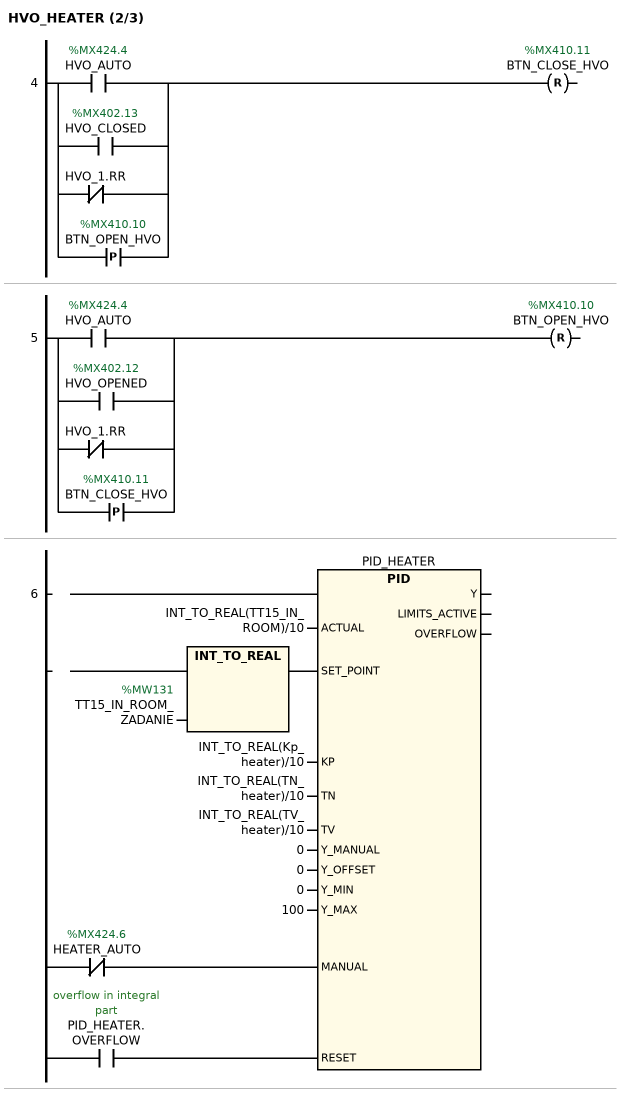
// NETWORK 4
//   HVO_AUTO: AT %MX424.4
//   HVO_CLOSED: AT %MX402.13
//   BTN_OPEN_HVO: AT %MX410.10
//   BTN_CLOSE_HVO: AT %MX410.11
_rt1(CLK := BTN_OPEN_HVO);
BTN_CLOSE_HVO R= HVO_AUTO OR HVO_CLOSED OR NOT HVO_1.RR OR _rt1.Q;

// NETWORK 5
//   HVO_AUTO: AT %MX424.4
//   HVO_OPENED: AT %MX402.12
//   BTN_CLOSE_HVO: AT %MX410.11
//   BTN_OPEN_HVO: AT %MX410.10
_rt2(CLK := BTN_CLOSE_HVO);
BTN_OPEN_HVO R= HVO_AUTO OR HVO_OPENED OR NOT HVO_1.RR OR _rt2.Q;

// NETWORK 6
//   TT15_IN_ROOM_ZADANIE: температура в комнате задание | AT %MW131
//   HEATER_AUTO: AT %MX424.6
//   PID_HEATER.OVERFLOW: overflow in integral part
PID_HEATER(
    ACTUAL := INT_TO_REAL(TT15_IN_ROOM)/10,
    SET_POINT := INT_TO_REAL(TT15_IN_ROOM_ZADANIE),
    KP := INT_TO_REAL(Kp_heater)/10,
    TN := INT_TO_REAL(TN_heater)/10,
    TV := INT_TO_REAL(TV_heater)/10,
    Y_MANUAL := 0,
    Y_OFFSET := 0,
    Y_MIN := 0,
    Y_MAX := 100,
    MANUAL := NOT HEATER_AUTO,
    RESET := PID_HEATER.OVERFLOW); // PID

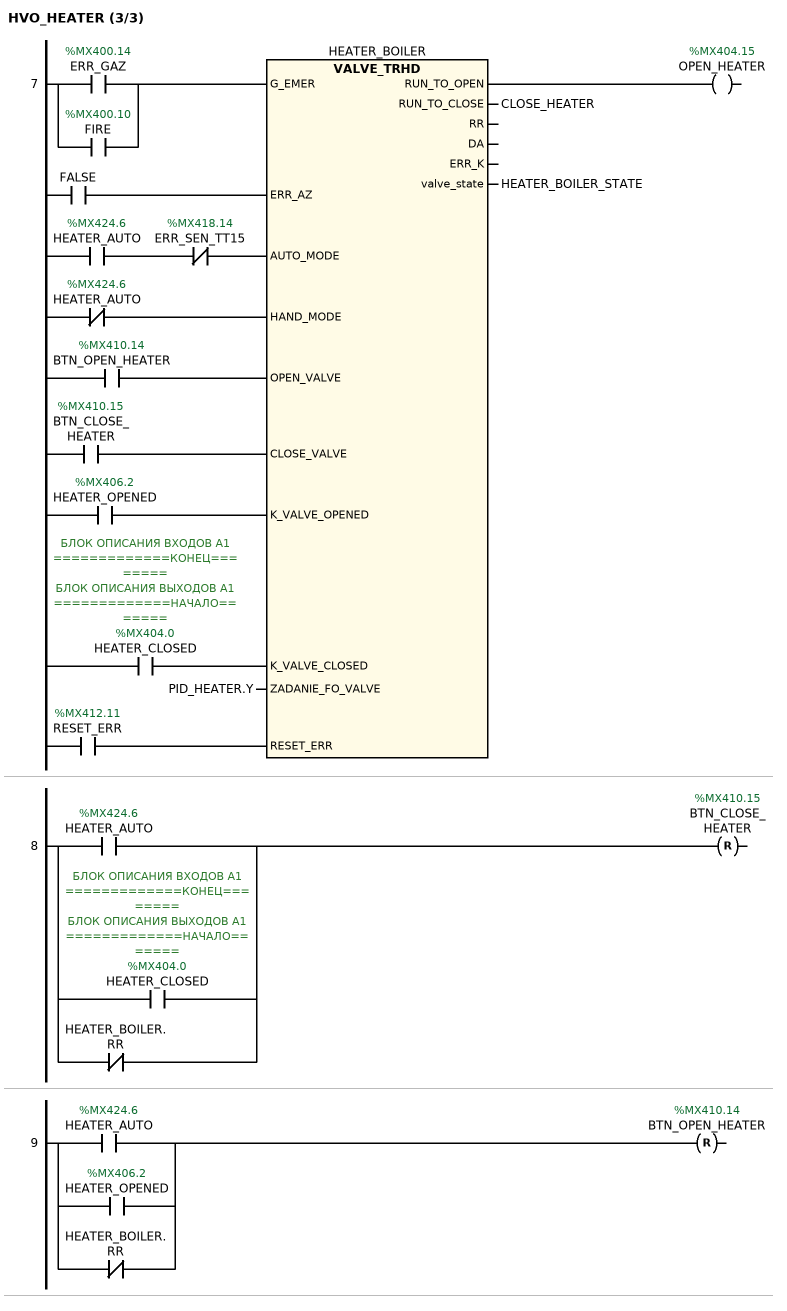
// NETWORK 7
//   ERR_GAZ: AT %MX400.14
//   FIRE: AT %MX400.10
//   HEATER_AUTO: AT %MX424.6
//   ERR_SEN_TT15: AT %MX418.14
//   BTN_OPEN_HEATER: AT %MX410.14
//   BTN_CLOSE_HEATER: AT %MX410.15
//   HEATER_OPENED: AT %MX406.2
//   HEATER_CLOSED: БЛОК ОПИСАНИЯ ВХОДОВ А1 =============КОНЕЦ======== БЛОК ОПИСАНИЯ ВЫХОДОВ А1 =============НАЧАЛО======= | AT %MX404.0
//   PID_HEATER.Y: manipulated variable, set value
//   RESET_ERR: AT %MX412.11
//   CLOSE_HEATER: AT %MX406.0
//   HEATER_BOILER_STATE: AT %MW404
//   OPEN_HEATER: AT %MX404.15
HEATER_BOILER(
    G_EMER := ERR_GAZ OR FIRE,
    ERR_AZ := FALSE,
    AUTO_MODE := HEATER_AUTO AND NOT ERR_SEN_TT15,
    HAND_MODE := NOT HEATER_AUTO,
    OPEN_VALVE := BTN_OPEN_HEATER,
    CLOSE_VALVE := BTN_CLOSE_HEATER,
    K_VALVE_OPENED := HEATER_OPENED,
    K_VALVE_CLOSED := HEATER_CLOSED,
    ZADANIE_FO_VALVE := PID_HEATER.Y,
    RESET_ERR := RESET_ERR,
    RUN_TO_CLOSE => CLOSE_HEATER,
    valve_state => HEATER_BOILER_STATE); // VALVE_TRHD
OPEN_HEATER := HEATER_BOILER.RUN_TO_OPEN;

// NETWORK 8
//   HEATER_AUTO: AT %MX424.6
//   HEATER_CLOSED: БЛОК ОПИСАНИЯ ВХОДОВ А1 =============КОНЕЦ======== БЛОК ОПИСАНИЯ ВЫХОДОВ А1 =============НАЧАЛО======= | AT %MX404.0
//   BTN_CLOSE_HEATER: AT %MX410.15
BTN_CLOSE_HEATER R= HEATER_AUTO OR HEATER_CLOSED OR NOT HEATER_BOILER.RR;

// NETWORK 9
//   HEATER_AUTO: AT %MX424.6
//   HEATER_OPENED: AT %MX406.2
//   BTN_OPEN_HEATER: AT %MX410.14
BTN_OPEN_HEATER R= HEATER_AUTO OR HEATER_OPENED OR NOT HEATER_BOILER.RR;

END_PROGRAM

// MyController/Application/FB/VALVE_TRHD
FUNCTION_BLOCK VALVE_TRHD
VAR_INPUT
	G_EMER: BOOL;
	ERR_AZ: BOOL;
	AUTO_MODE: BOOL;
	HAND_MODE: BOOL;
	OPEN_VALVE: BOOL;
	CLOSE_VALVE: BOOL;
	K_VALVE_OPENED: BOOL;
	K_VALVE_CLOSED: BOOL;
	ZADANIE_FO_VALVE: REAL;
	RESET_ERR: BOOL;	
END_VAR
VAR_OUTPUT
	RUN_TO_OPEN: BOOL;
	RUN_TO_CLOSE: BOOL;
	RR: BOOL;
	DA: BOOL;
	ERR_K: BOOL;
	valve_state: BYTE;
END_VAR
VAR
	TM_LT_VALVE: TON;
	RUN_VALVE_TO_OPEN: BOOL;
	CYCLE_OPEN: BOOL;
	CYCLE_CLOSE: BOOL;
END_VAR
VAR // added by the converter: edge detectors and wires of the graphical bodies
    _w1 : BOOL;
END_VAR

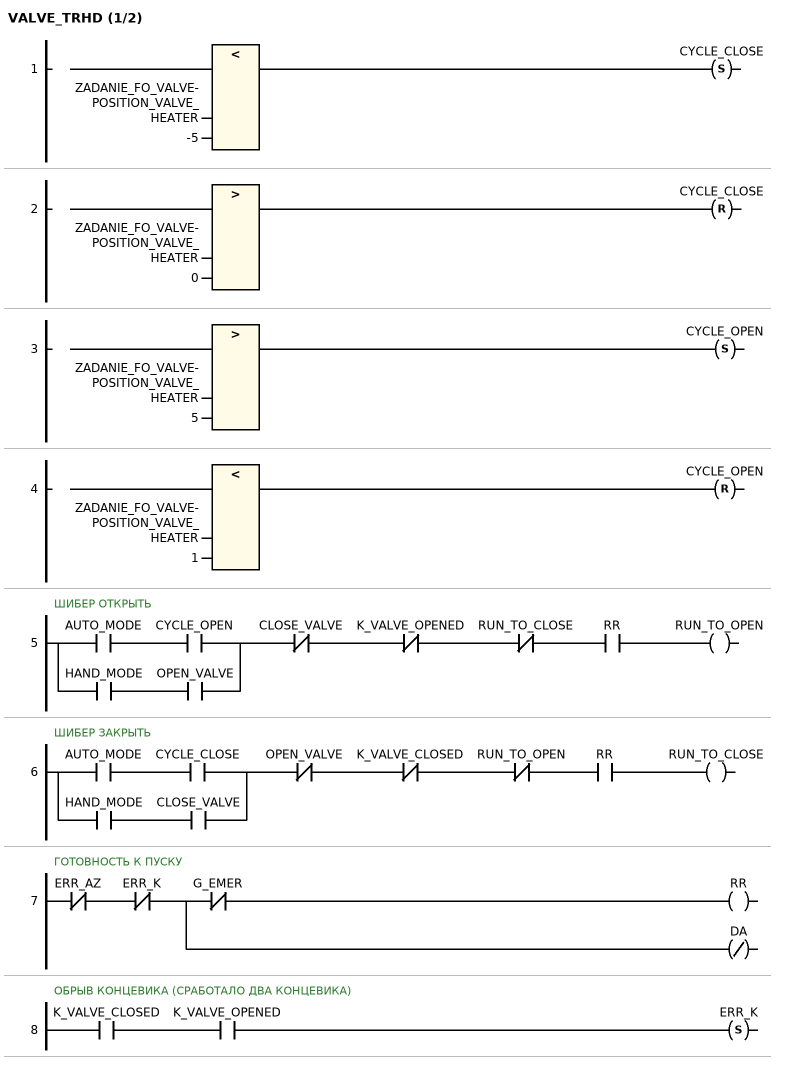
// NETWORK 1
CYCLE_CLOSE S= (ZADANIE_FO_VALVE-POSITION_VALVE_HEATER) < -5;

// NETWORK 2
CYCLE_CLOSE R= (ZADANIE_FO_VALVE-POSITION_VALVE_HEATER) > 0;

// NETWORK 3
CYCLE_OPEN S= (ZADANIE_FO_VALVE-POSITION_VALVE_HEATER) > 5;

// NETWORK 4
CYCLE_OPEN R= (ZADANIE_FO_VALVE-POSITION_VALVE_HEATER) < 1;

// NETWORK 5
// ШИБЕР ОТКРЫТЬ
RUN_TO_OPEN := (AUTO_MODE AND CYCLE_OPEN OR HAND_MODE AND OPEN_VALVE) AND NOT CLOSE_VALVE AND NOT K_VALVE_OPENED AND NOT RUN_TO_CLOSE AND RR;

// NETWORK 6
// ШИБЕР ЗАКРЫТЬ
RUN_TO_CLOSE := (AUTO_MODE AND CYCLE_CLOSE OR HAND_MODE AND CLOSE_VALVE) AND NOT OPEN_VALVE AND NOT K_VALVE_CLOSED AND NOT RUN_TO_OPEN AND RR;

// NETWORK 7
// ГОТОВНОСТЬ К ПУСКУ
_w1 := NOT ERR_AZ AND NOT ERR_K;
RR := _w1 AND NOT G_EMER;
DA := NOT _w1;

// NETWORK 8
// ОБРЫВ КОНЦЕВИКА (СРАБОТАЛО ДВА КОНЦЕВИКА)
ERR_K S= K_VALVE_CLOSED AND K_VALVE_OPENED;

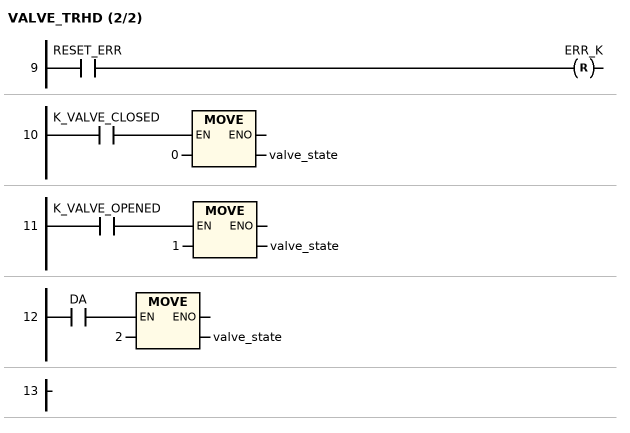
// NETWORK 9
ERR_K R= RESET_ERR;

// NETWORK 10
IF K_VALVE_CLOSED THEN valve_state := 0; END_IF

// NETWORK 11
IF K_VALVE_OPENED THEN valve_state := 1; END_IF

// NETWORK 12
IF DA THEN valve_state := 2; END_IF

// NETWORK 13

END_FUNCTION_BLOCK

// MyController/Application/connection
PROGRAM connection
VAR
	connection_off: TON;
	set_connection: BLINK;
	tm_connection: TON;
END_VAR
VAR // added by the converter: edge detectors and wires of the graphical bodies
    _rt1, _rt2 : R_TRIG;
END_VAR

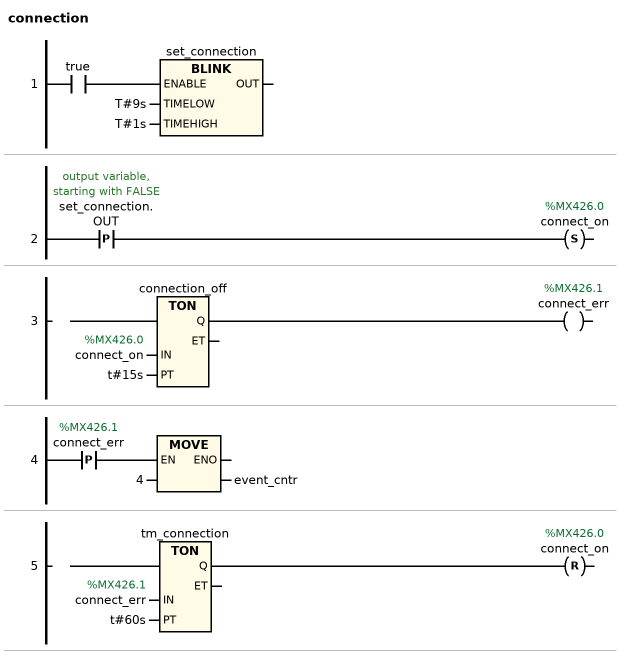
// NETWORK 1
set_connection(ENABLE := true, TIMELOW := T#9s, TIMEHIGH := T#1s); // BLINK

// NETWORK 2
//   set_connection.OUT: output variable, starting with FALSE
//   connect_on: AT %MX426.0
_rt1(CLK := set_connection.OUT);
connect_on S= _rt1.Q;

// NETWORK 3
//   connect_on: AT %MX426.0
//   connect_err: AT %MX426.1
connection_off(IN := connect_on, PT := t#15s); // TON
connect_err := connection_off.Q;

// NETWORK 4
//   connect_err: AT %MX426.1
//   event_cntr: AT %MW986
_rt2(CLK := connect_err);
IF _rt2.Q THEN event_cntr := 4; END_IF

// NETWORK 5
//   connect_err: AT %MX426.1
//   connect_on: AT %MX426.0
tm_connection(IN := connect_err, PT := t#60s); // TON
connect_on R= tm_connection.Q;

END_PROGRAM

// MyController/Application/DYMOHODS
PROGRAM DYMOHODS
VAR
	STOP_DYMOHOD_1: TON;
	STOP_DYMOHOD_2: TON;
END_VAR
VAR // added by the converter: edge detectors and wires of the graphical bodies
    _rt1, _rt2, _rt3, _rt4 : R_TRIG;
END_VAR

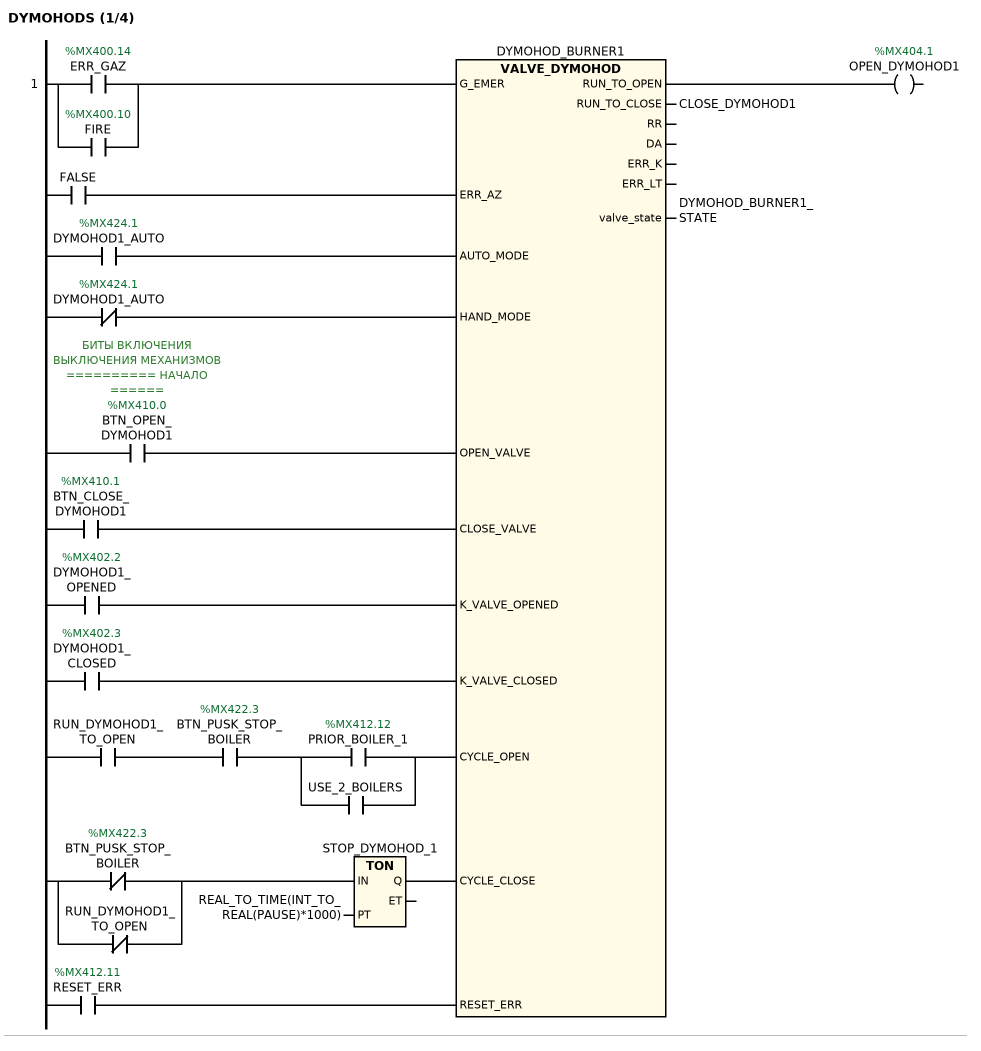
// NETWORK 1
//   ERR_GAZ: AT %MX400.14
//   FIRE: AT %MX400.10
//   DYMOHOD1_AUTO: AT %MX424.1
//   BTN_OPEN_DYMOHOD1: БИТЫ ВКЛЮЧЕНИЯ ВЫКЛЮЧЕНИЯ МЕХАНИЗМОВ ========== НАЧАЛО ====== | AT %MX410.0
//   BTN_CLOSE_DYMOHOD1: AT %MX410.1
//   DYMOHOD1_OPENED: AT %MX402.2
//   DYMOHOD1_CLOSED: AT %MX402.3
//   BTN_PUSK_STOP_BOILER: AT %MX422.3
//   PRIOR_BOILER_1: AT %MX412.12
//   RESET_ERR: AT %MX412.11
//   CLOSE_DYMOHOD1: AT %MX404.2
//   DYMOHOD_BURNER1_STATE: AT %MW401
//   OPEN_DYMOHOD1: AT %MX404.1
STOP_DYMOHOD_1(IN := NOT BTN_PUSK_STOP_BOILER OR NOT RUN_DYMOHOD1_TO_OPEN, PT := REAL_TO_TIME(INT_TO_REAL(PAUSE)*1000)); // TON
DYMOHOD_BURNER1(
    G_EMER := ERR_GAZ OR FIRE,
    ERR_AZ := FALSE,
    AUTO_MODE := DYMOHOD1_AUTO,
    HAND_MODE := NOT DYMOHOD1_AUTO,
    OPEN_VALVE := BTN_OPEN_DYMOHOD1,
    CLOSE_VALVE := BTN_CLOSE_DYMOHOD1,
    K_VALVE_OPENED := DYMOHOD1_OPENED,
    K_VALVE_CLOSED := DYMOHOD1_CLOSED,
    CYCLE_OPEN := RUN_DYMOHOD1_TO_OPEN AND BTN_PUSK_STOP_BOILER AND (PRIOR_BOILER_1 OR USE_2_BOILERS),
    CYCLE_CLOSE := STOP_DYMOHOD_1.Q,
    RESET_ERR := RESET_ERR,
    RUN_TO_CLOSE => CLOSE_DYMOHOD1,
    valve_state => DYMOHOD_BURNER1_STATE); // VALVE_DYMOHOD
OPEN_DYMOHOD1 := DYMOHOD_BURNER1.RUN_TO_OPEN;

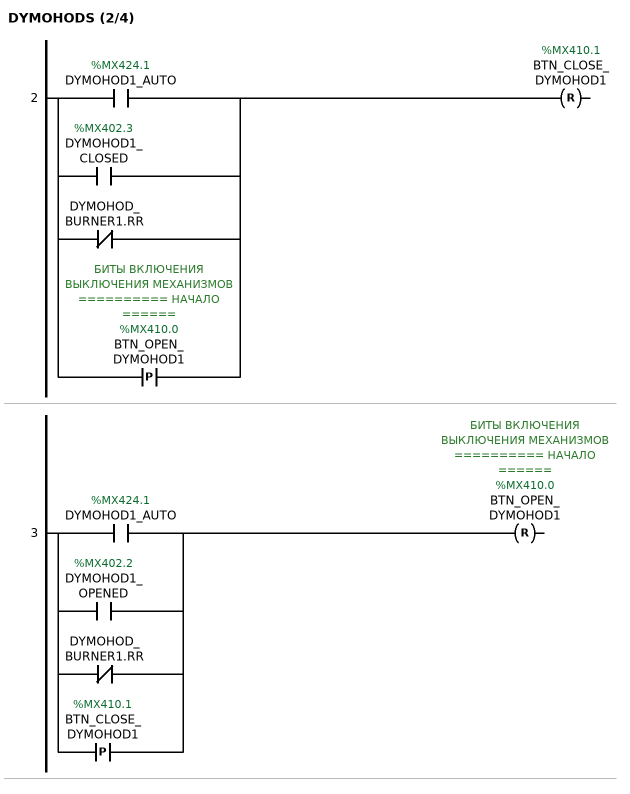
// NETWORK 2
//   DYMOHOD1_AUTO: AT %MX424.1
//   DYMOHOD1_CLOSED: AT %MX402.3
//   BTN_OPEN_DYMOHOD1: БИТЫ ВКЛЮЧЕНИЯ ВЫКЛЮЧЕНИЯ МЕХАНИЗМОВ ========== НАЧАЛО ====== | AT %MX410.0
//   BTN_CLOSE_DYMOHOD1: AT %MX410.1
_rt1(CLK := BTN_OPEN_DYMOHOD1);
BTN_CLOSE_DYMOHOD1 R= DYMOHOD1_AUTO OR DYMOHOD1_CLOSED OR NOT DYMOHOD_BURNER1.RR OR _rt1.Q;

// NETWORK 3
//   DYMOHOD1_AUTO: AT %MX424.1
//   DYMOHOD1_OPENED: AT %MX402.2
//   BTN_CLOSE_DYMOHOD1: AT %MX410.1
//   BTN_OPEN_DYMOHOD1: БИТЫ ВКЛЮЧЕНИЯ ВЫКЛЮЧЕНИЯ МЕХАНИЗМОВ ========== НАЧАЛО ====== | AT %MX410.0
_rt2(CLK := BTN_CLOSE_DYMOHOD1);
BTN_OPEN_DYMOHOD1 R= DYMOHOD1_AUTO OR DYMOHOD1_OPENED OR NOT DYMOHOD_BURNER1.RR OR _rt2.Q;

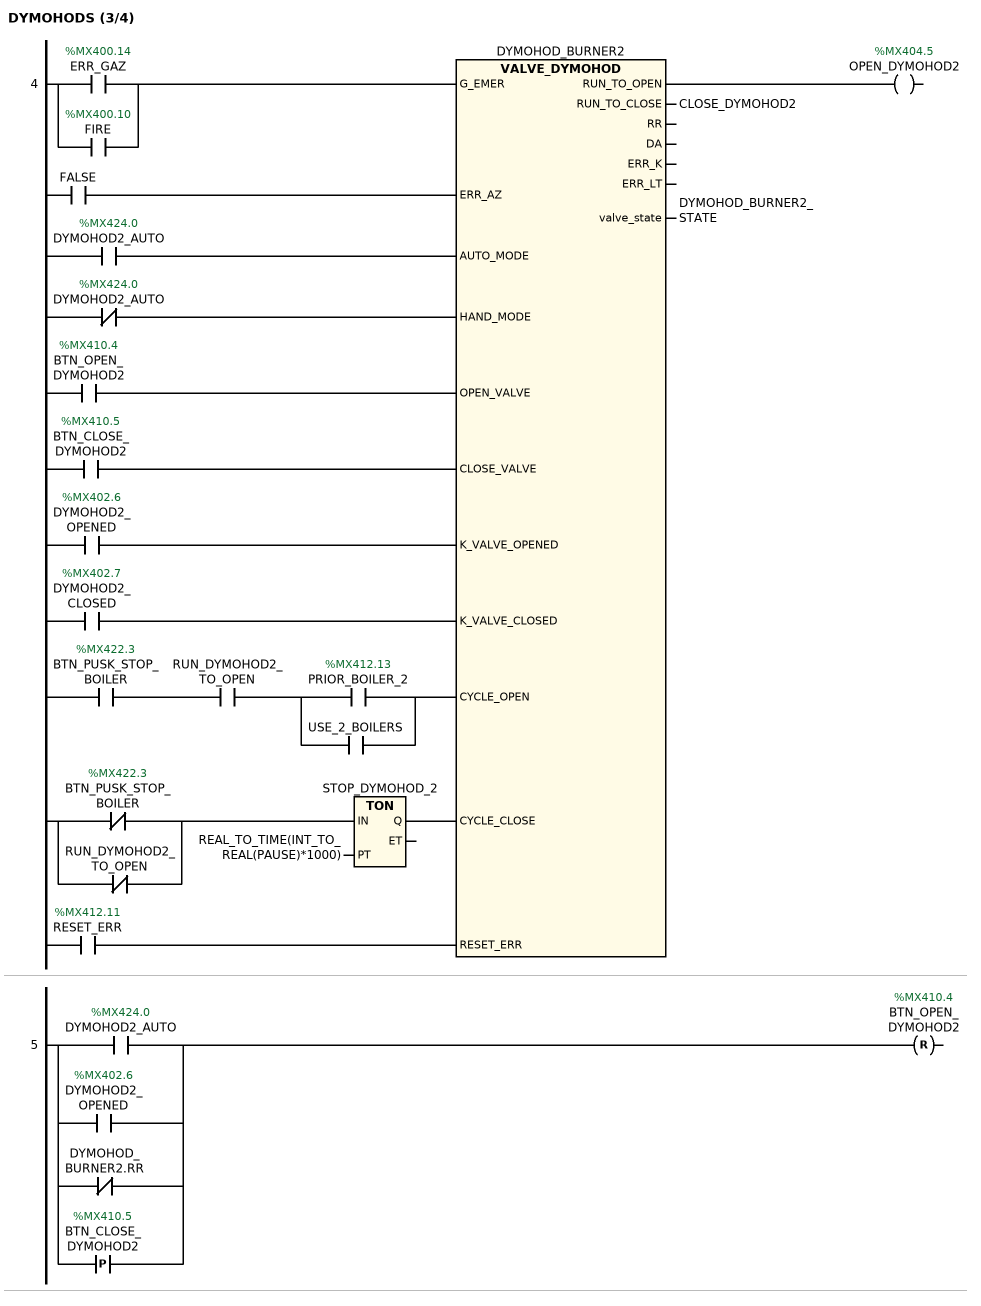
// NETWORK 4
//   ERR_GAZ: AT %MX400.14
//   FIRE: AT %MX400.10
//   DYMOHOD2_AUTO: AT %MX424.0
//   BTN_OPEN_DYMOHOD2: AT %MX410.4
//   BTN_CLOSE_DYMOHOD2: AT %MX410.5
//   DYMOHOD2_OPENED: AT %MX402.6
//   DYMOHOD2_CLOSED: AT %MX402.7
//   BTN_PUSK_STOP_BOILER: AT %MX422.3
//   PRIOR_BOILER_2: AT %MX412.13
//   RESET_ERR: AT %MX412.11
//   CLOSE_DYMOHOD2: AT %MX404.6
//   DYMOHOD_BURNER2_STATE: AT %MW402
//   OPEN_DYMOHOD2: AT %MX404.5
STOP_DYMOHOD_2(IN := NOT BTN_PUSK_STOP_BOILER OR NOT RUN_DYMOHOD2_TO_OPEN, PT := REAL_TO_TIME(INT_TO_REAL(PAUSE)*1000)); // TON
DYMOHOD_BURNER2(
    G_EMER := ERR_GAZ OR FIRE,
    ERR_AZ := FALSE,
    AUTO_MODE := DYMOHOD2_AUTO,
    HAND_MODE := NOT DYMOHOD2_AUTO,
    OPEN_VALVE := BTN_OPEN_DYMOHOD2,
    CLOSE_VALVE := BTN_CLOSE_DYMOHOD2,
    K_VALVE_OPENED := DYMOHOD2_OPENED,
    K_VALVE_CLOSED := DYMOHOD2_CLOSED,
    CYCLE_OPEN := BTN_PUSK_STOP_BOILER AND RUN_DYMOHOD2_TO_OPEN AND (PRIOR_BOILER_2 OR USE_2_BOILERS),
    CYCLE_CLOSE := STOP_DYMOHOD_2.Q,
    RESET_ERR := RESET_ERR,
    RUN_TO_CLOSE => CLOSE_DYMOHOD2,
    valve_state => DYMOHOD_BURNER2_STATE); // VALVE_DYMOHOD
OPEN_DYMOHOD2 := DYMOHOD_BURNER2.RUN_TO_OPEN;

// NETWORK 5
//   DYMOHOD2_AUTO: AT %MX424.0
//   DYMOHOD2_OPENED: AT %MX402.6
//   BTN_CLOSE_DYMOHOD2: AT %MX410.5
//   BTN_OPEN_DYMOHOD2: AT %MX410.4
_rt3(CLK := BTN_CLOSE_DYMOHOD2);
BTN_OPEN_DYMOHOD2 R= DYMOHOD2_AUTO OR DYMOHOD2_OPENED OR NOT DYMOHOD_BURNER2.RR OR _rt3.Q;

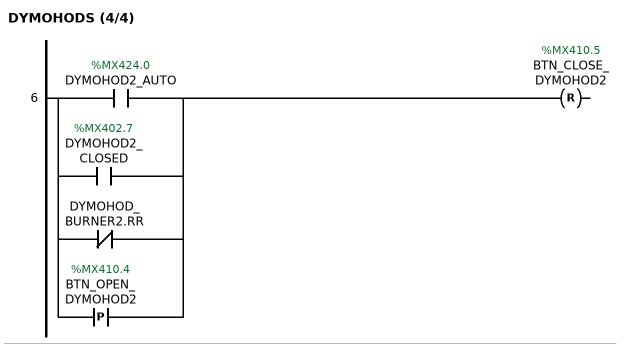
// NETWORK 6
//   DYMOHOD2_AUTO: AT %MX424.0
//   DYMOHOD2_CLOSED: AT %MX402.7
//   BTN_OPEN_DYMOHOD2: AT %MX410.4
//   BTN_CLOSE_DYMOHOD2: AT %MX410.5
_rt4(CLK := BTN_OPEN_DYMOHOD2);
BTN_CLOSE_DYMOHOD2 R= DYMOHOD2_AUTO OR DYMOHOD2_CLOSED OR NOT DYMOHOD_BURNER2.RR OR _rt4.Q;

END_PROGRAM

// MyController/Application/FB/VALVE_DYMOHOD
FUNCTION_BLOCK VALVE_DYMOHOD
VAR_INPUT
	G_EMER: BOOL;
	ERR_AZ: BOOL;
	AUTO_MODE: BOOL;
	HAND_MODE: BOOL;
	OPEN_VALVE: BOOL;
	CLOSE_VALVE: BOOL;
	K_VALVE_OPENED: BOOL;
	K_VALVE_CLOSED: BOOL;
	CYCLE_OPEN: BOOL;
	CYCLE_CLOSE: BOOL;
	RESET_ERR: BOOL;	
END_VAR
VAR_OUTPUT
	RUN_TO_OPEN: BOOL;
	RUN_TO_CLOSE: BOOL;
	RR: BOOL;
	DA: BOOL;
	ERR_K: BOOL;
	ERR_LT: BOOL;
	valve_state: BYTE;
END_VAR
VAR
	TM_LT_VALVE: TON;
END_VAR
VAR // added by the converter: edge detectors and wires of the graphical bodies
    _w1 : BOOL;
END_VAR

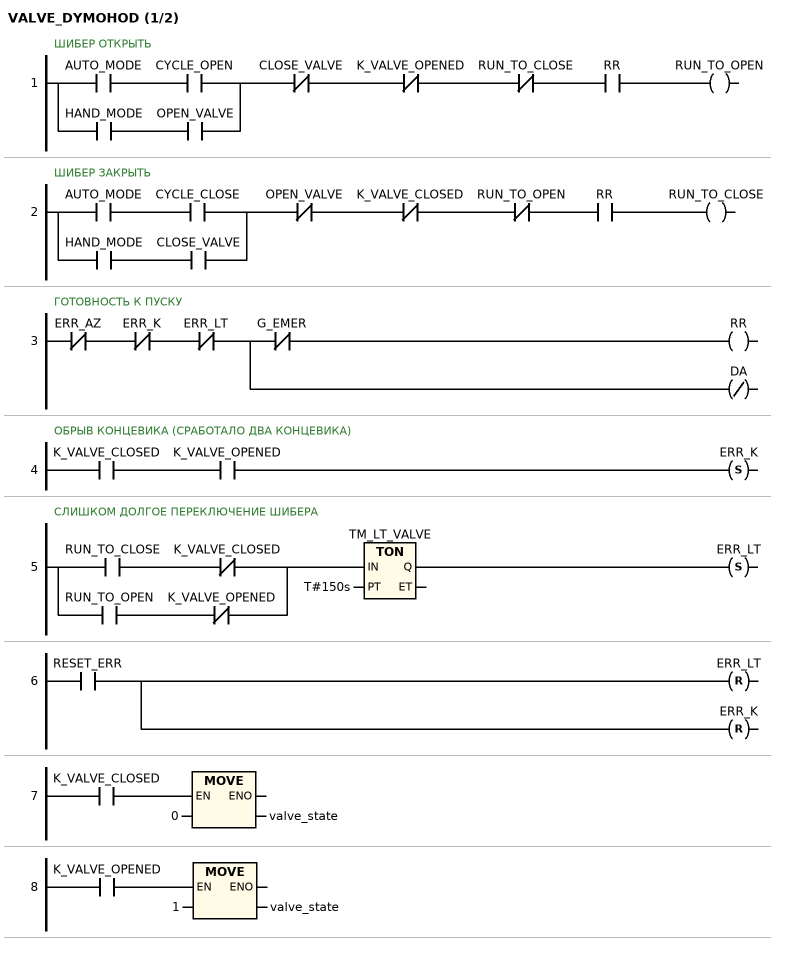
// NETWORK 1
// ШИБЕР ОТКРЫТЬ
RUN_TO_OPEN := (AUTO_MODE AND CYCLE_OPEN OR HAND_MODE AND OPEN_VALVE) AND NOT CLOSE_VALVE AND NOT K_VALVE_OPENED AND NOT RUN_TO_CLOSE AND RR;

// NETWORK 2
// ШИБЕР ЗАКРЫТЬ
RUN_TO_CLOSE := (AUTO_MODE AND CYCLE_CLOSE OR HAND_MODE AND CLOSE_VALVE) AND NOT OPEN_VALVE AND NOT K_VALVE_CLOSED AND NOT RUN_TO_OPEN AND RR;

// NETWORK 3
// ГОТОВНОСТЬ К ПУСКУ
_w1 := NOT ERR_AZ AND NOT ERR_K AND NOT ERR_LT;
RR := _w1 AND NOT G_EMER;
DA := NOT _w1;

// NETWORK 4
// ОБРЫВ КОНЦЕВИКА (СРАБОТАЛО ДВА КОНЦЕВИКА)
ERR_K S= K_VALVE_CLOSED AND K_VALVE_OPENED;

// NETWORK 5
// СЛИШКОМ ДОЛГОЕ ПЕРЕКЛЮЧЕНИЕ ШИБЕРА
TM_LT_VALVE(IN := RUN_TO_CLOSE AND NOT K_VALVE_CLOSED OR RUN_TO_OPEN AND NOT K_VALVE_OPENED, PT := T#150s); // TON
ERR_LT S= TM_LT_VALVE.Q;

// NETWORK 6
ERR_LT R= RESET_ERR;
ERR_K R= RESET_ERR;

// NETWORK 7
IF K_VALVE_CLOSED THEN valve_state := 0; END_IF

// NETWORK 8
IF K_VALVE_OPENED THEN valve_state := 1; END_IF

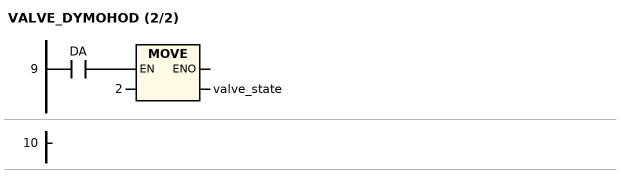
// NETWORK 9
IF DA THEN valve_state := 2; END_IF

// NETWORK 10

END_FUNCTION_BLOCK

// MyController/Application/RECIRCULATIONS_M5_M6_M7
PROGRAM RECIRCULATIONS_M5_M6_M7
VAR
	PUMP_M5_CYCLE: BOOL;
	PUMP_M6_CYCLE: BOOL;
	PUMP_M7_CYCLE: BOOL;
	PID_M7: PID;
END_VAR

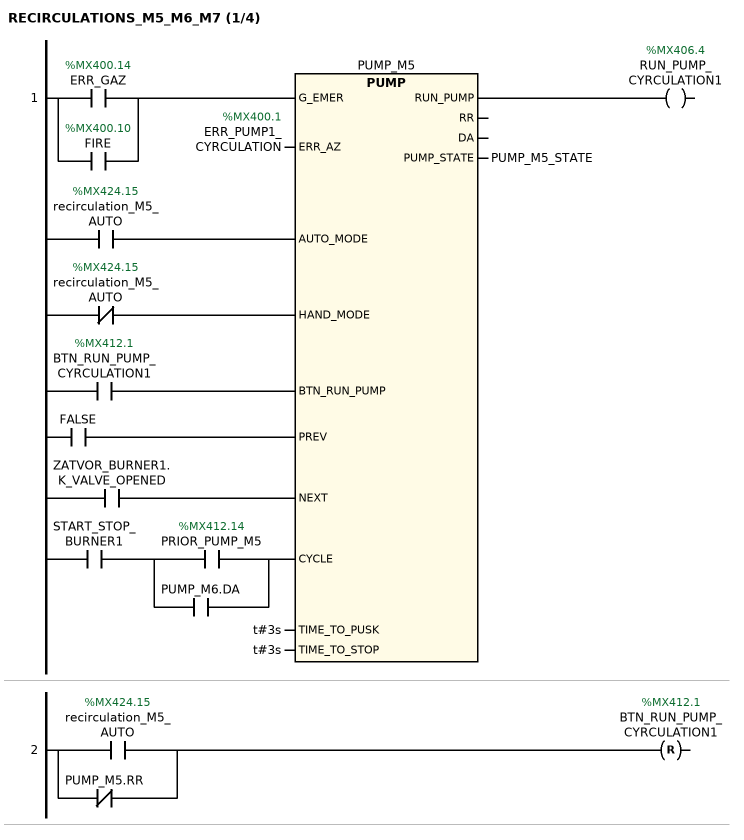
// NETWORK 1
//   ERR_GAZ: AT %MX400.14
//   FIRE: AT %MX400.10
//   ERR_PUMP1_CYRCULATION: AT %MX400.1
//   recirculation_M5_AUTO: AT %MX424.15
//   BTN_RUN_PUMP_CYRCULATION1: AT %MX412.1
//   PRIOR_PUMP_M5: AT %MX412.14
//   PUMP_M5_STATE: AT %MW413
//   RUN_PUMP_CYRCULATION1: AT %MX406.4
PUMP_M5(
    G_EMER := ERR_GAZ OR FIRE,
    ERR_AZ := ERR_PUMP1_CYRCULATION,
    AUTO_MODE := recirculation_M5_AUTO,
    HAND_MODE := NOT recirculation_M5_AUTO,
    BTN_RUN_PUMP := BTN_RUN_PUMP_CYRCULATION1,
    PREV := FALSE,
    NEXT := ZATVOR_BURNER1.K_VALVE_OPENED,
    CYCLE := START_STOP_BURNER1 AND (PRIOR_PUMP_M5 OR PUMP_M6.DA),
    TIME_TO_PUSK := t#3s,
    TIME_TO_STOP := t#3s,
    PUMP_STATE => PUMP_M5_STATE); // PUMP
RUN_PUMP_CYRCULATION1 := PUMP_M5.RUN_PUMP;

// NETWORK 2
//   recirculation_M5_AUTO: AT %MX424.15
//   BTN_RUN_PUMP_CYRCULATION1: AT %MX412.1
BTN_RUN_PUMP_CYRCULATION1 R= recirculation_M5_AUTO OR NOT PUMP_M5.RR;

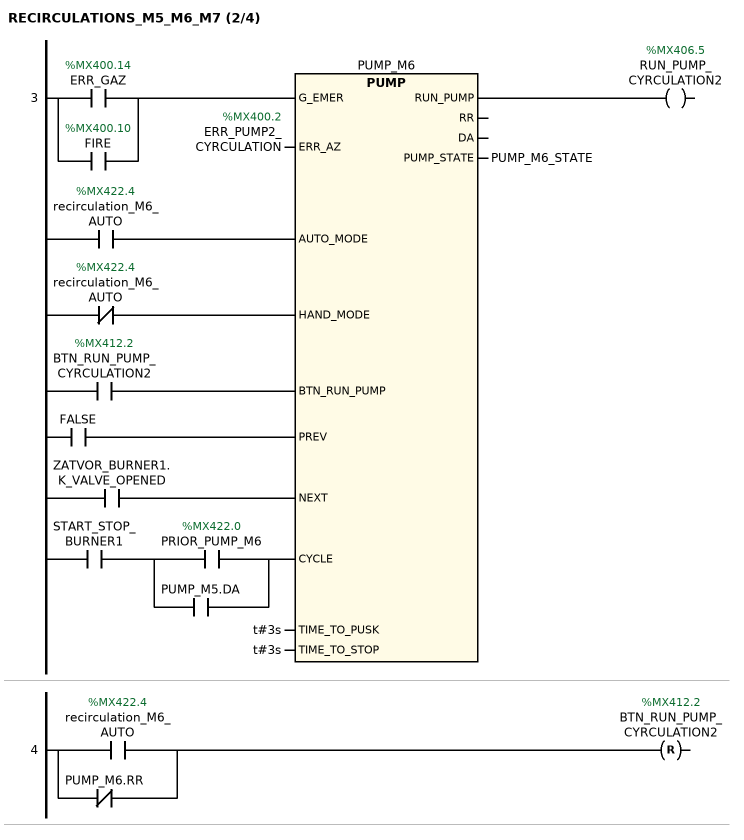
// NETWORK 3
//   ERR_GAZ: AT %MX400.14
//   FIRE: AT %MX400.10
//   ERR_PUMP2_CYRCULATION: AT %MX400.2
//   recirculation_M6_AUTO: AT %MX422.4
//   BTN_RUN_PUMP_CYRCULATION2: AT %MX412.2
//   PRIOR_PUMP_M6: AT %MX422.0
//   PUMP_M6_STATE: AT %MW414
//   RUN_PUMP_CYRCULATION2: AT %MX406.5
PUMP_M6(
    G_EMER := ERR_GAZ OR FIRE,
    ERR_AZ := ERR_PUMP2_CYRCULATION,
    AUTO_MODE := recirculation_M6_AUTO,
    HAND_MODE := NOT recirculation_M6_AUTO,
    BTN_RUN_PUMP := BTN_RUN_PUMP_CYRCULATION2,
    PREV := FALSE,
    NEXT := ZATVOR_BURNER1.K_VALVE_OPENED,
    CYCLE := START_STOP_BURNER1 AND (PRIOR_PUMP_M6 OR PUMP_M5.DA),
    TIME_TO_PUSK := t#3s,
    TIME_TO_STOP := t#3s,
    PUMP_STATE => PUMP_M6_STATE); // PUMP
RUN_PUMP_CYRCULATION2 := PUMP_M6.RUN_PUMP;

// NETWORK 4
//   recirculation_M6_AUTO: AT %MX422.4
//   BTN_RUN_PUMP_CYRCULATION2: AT %MX412.2
BTN_RUN_PUMP_CYRCULATION2 R= recirculation_M6_AUTO OR NOT PUMP_M6.RR;

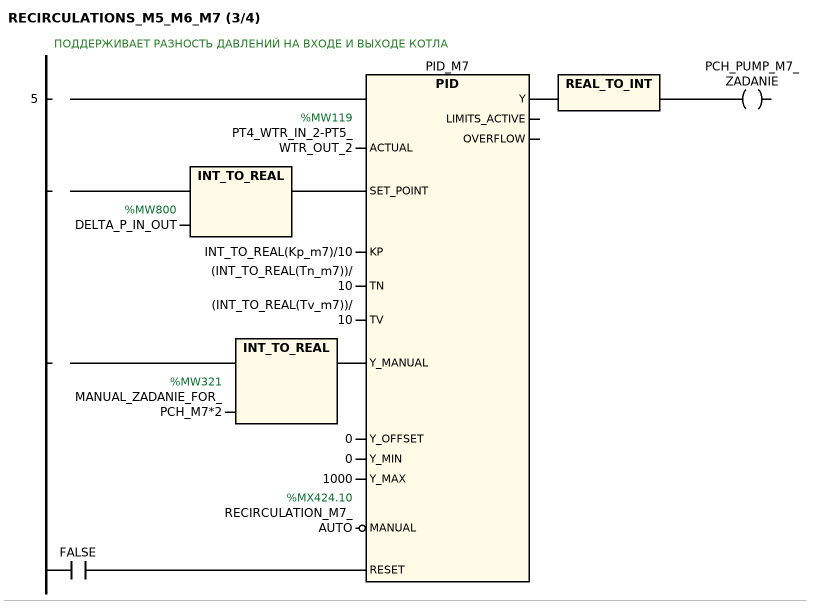
// NETWORK 5
// ПОДДЕРЖИВАЕТ РАЗНОСТЬ ДАВЛЕНИЙ НА ВХОДЕ И ВЫХОДЕ КОТЛА
//   PT4_WTR_IN_2-PT5_WTR_OUT_2: AT %MW119
//   DELTA_P_IN_OUT: AT %MW800
//   MANUAL_ZADANIE_FOR_PCH_M7*2: AT %MW321
//   RECIRCULATION_M7_AUTO: AT %MX424.10
PID_M7(
    ACTUAL := PT4_WTR_IN_2-PT5_WTR_OUT_2,
    SET_POINT := INT_TO_REAL(DELTA_P_IN_OUT),
    KP := INT_TO_REAL(Kp_m7)/10,
    TN := (INT_TO_REAL(Tn_m7))/10,
    TV := (INT_TO_REAL(Tv_m7))/10,
    Y_MANUAL := INT_TO_REAL(MANUAL_ZADANIE_FOR_PCH_M7*2),
    Y_OFFSET := 0,
    Y_MIN := 0,
    Y_MAX := 1000,
    MANUAL := NOT RECIRCULATION_M7_AUTO,
    RESET := FALSE); // PID
PCH_PUMP_M7_ZADANIE := REAL_TO_INT(PID_M7.Y);

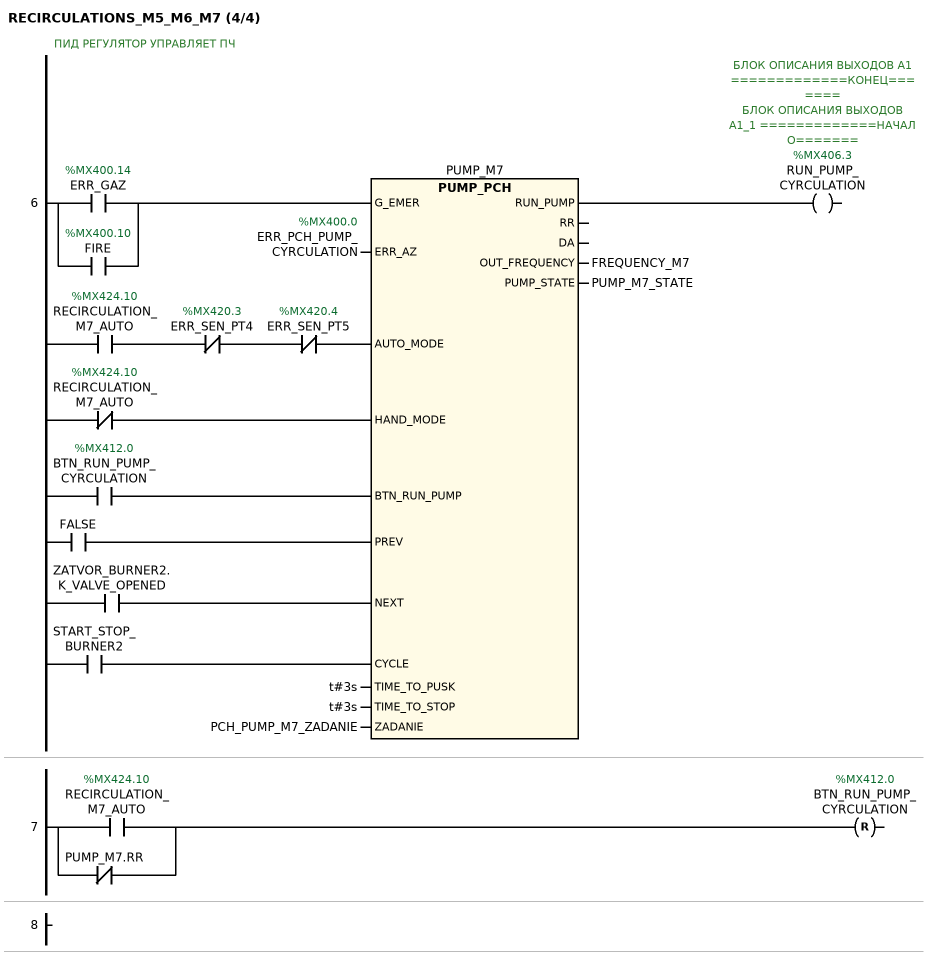
// NETWORK 6
// ПИД РЕГУЛЯТОР УПРАВЛЯЕТ ПЧ
//   ERR_GAZ: AT %MX400.14
//   FIRE: AT %MX400.10
//   ERR_PCH_PUMP_CYRCULATION: БЛОК ДЛЯ ОБМЕНА С ОВЕНОМ ======КОЕЦ====== БЛОК ОПИСАНИЯ ВХОДОВ А1_1 A1_2 =============НАЧАЛО======= | AT %MX400.0
//   RECIRCULATION_M7_AUTO: AT %MX424.10
//   ERR_SEN_PT4: AT %MX420.3
//   ERR_SEN_PT5: AT %MX420.4
//   BTN_RUN_PUMP_CYRCULATION: AT %MX412.0
//   FREQUENCY_M7: AT %MW136
//   PUMP_M7_STATE: AT %MW415
//   RUN_PUMP_CYRCULATION: БЛОК ОПИСАНИЯ ВЫХОДОВ А1 =============КОНЕЦ======= БЛОК ОПИСАНИЯ ВЫХОДОВ А1_1 =============НАЧАЛО======= | AT %MX406.3
PUMP_M7(
    G_EMER := ERR_GAZ OR FIRE,
    ERR_AZ := ERR_PCH_PUMP_CYRCULATION,
    AUTO_MODE := RECIRCULATION_M7_AUTO AND NOT ERR_SEN_PT4 AND NOT ERR_SEN_PT5,
    HAND_MODE := NOT RECIRCULATION_M7_AUTO,
    BTN_RUN_PUMP := BTN_RUN_PUMP_CYRCULATION,
    PREV := FALSE,
    NEXT := ZATVOR_BURNER2.K_VALVE_OPENED,
    CYCLE := START_STOP_BURNER2,
    TIME_TO_PUSK := t#3s,
    TIME_TO_STOP := t#3s,
    ZADANIE := PCH_PUMP_M7_ZADANIE,
    OUT_FREQUENCY => FREQUENCY_M7,
    PUMP_STATE => PUMP_M7_STATE); // PUMP_PCH
RUN_PUMP_CYRCULATION := PUMP_M7.RUN_PUMP;

// NETWORK 7
//   RECIRCULATION_M7_AUTO: AT %MX424.10
//   BTN_RUN_PUMP_CYRCULATION: AT %MX412.0
BTN_RUN_PUMP_CYRCULATION R= RECIRCULATION_M7_AUTO OR NOT PUMP_M7.RR;

// NETWORK 8

END_PROGRAM

// MyController/Application/FB/PUMP
FUNCTION_BLOCK PUMP
VAR_INPUT
	G_EMER: BOOL;
	ERR_AZ: BOOL;		
	AUTO_MODE: BOOL;
	HAND_MODE: BOOL;
	BTN_RUN_PUMP: BOOL;
	PREV: BOOL;
	NEXT: BOOL;	
	CYCLE: BOOL;	
	TIME_TO_PUSK: TIME;
	TIME_TO_STOP: TIME;		
END_VAR
VAR_OUTPUT
	RUN_PUMP: BOOL;
	RR: BOOL;
	DA: BOOL;	
	PUMP_STATE: BYTE;
END_VAR
VAR
	AUTO: BOOL;
	TM_PUSK_PUMP: TON;
	TM_STOP_PUMP: TON;
END_VAR
VAR // added by the converter: edge detectors and wires of the graphical bodies
    _w1 : BOOL;
END_VAR

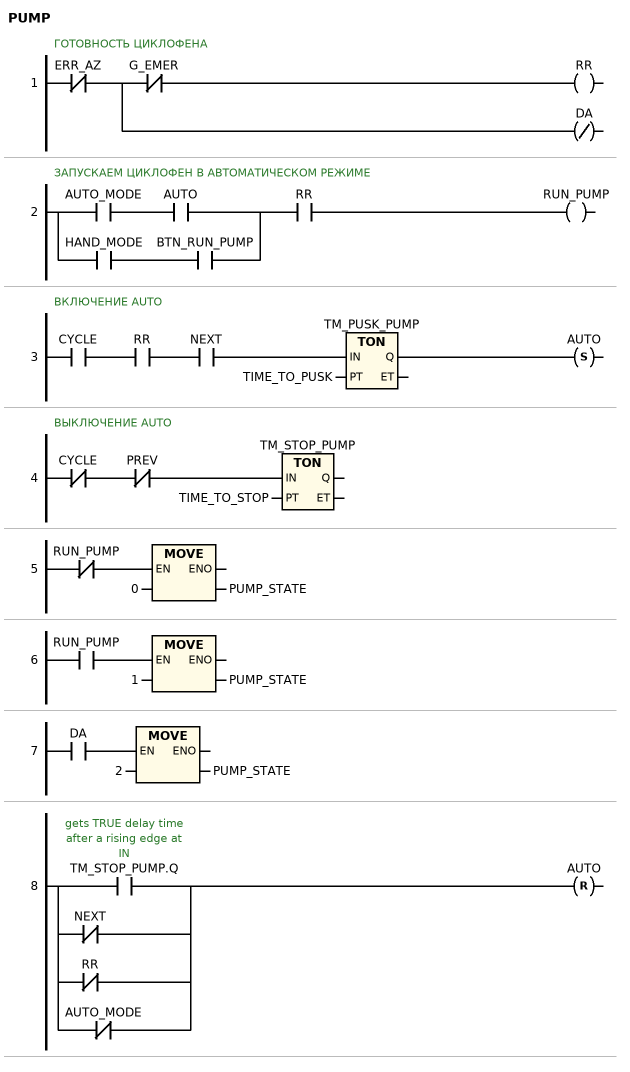
// NETWORK 1
// ГОТОВНОСТЬ ЦИКЛОФЕНА
_w1 := NOT ERR_AZ;
RR := _w1 AND NOT G_EMER;
DA := NOT _w1;

// NETWORK 2
// ЗАПУСКАЕМ ЦИКЛОФЕН В АВТОМАТИЧЕСКОМ РЕЖИМЕ
RUN_PUMP := (AUTO_MODE AND AUTO OR HAND_MODE AND BTN_RUN_PUMP) AND RR;

// NETWORK 3
// ВКЛЮЧЕНИЕ AUTO
TM_PUSK_PUMP(IN := CYCLE AND RR AND NEXT, PT := TIME_TO_PUSK); // TON
AUTO S= TM_PUSK_PUMP.Q;

// NETWORK 4
// ВЫКЛЮЧЕНИЕ AUTO
TM_STOP_PUMP(IN := NOT CYCLE AND NOT PREV, PT := TIME_TO_STOP); // TON

// NETWORK 5
IF NOT RUN_PUMP THEN PUMP_STATE := 0; END_IF

// NETWORK 6
IF RUN_PUMP THEN PUMP_STATE := 1; END_IF

// NETWORK 7
IF DA THEN PUMP_STATE := 2; END_IF

// NETWORK 8
//   TM_STOP_PUMP.Q: gets TRUE delay time after a rising edge at IN
AUTO R= TM_STOP_PUMP.Q OR NOT NEXT OR NOT RR OR NOT AUTO_MODE;

END_FUNCTION_BLOCK

// MyController/Application/FB/PUMP_PCH
FUNCTION_BLOCK PUMP_PCH
VAR_INPUT
	G_EMER: BOOL;
	ERR_AZ: BOOL;		
	AUTO_MODE: BOOL;
	HAND_MODE: BOOL;
	BTN_RUN_PUMP: BOOL;
	PREV: BOOL;
	NEXT: BOOL;	
	CYCLE: BOOL;	
	TIME_TO_PUSK: TIME;
	TIME_TO_STOP: TIME;		
	ZADANIE: INT;
END_VAR
VAR_OUTPUT
	RUN_PUMP: BOOL;
	RR: BOOL;
	DA: BOOL;	
	OUT_FREQUENCY: INT;
	PUMP_STATE: BYTE;
END_VAR
VAR
	AUTO: BOOL;
	TM_PUSK_PUMP: TON;
	TM_STOP_PUMP: TON;
END_VAR
VAR // added by the converter: edge detectors and wires of the graphical bodies
    _w1 : BOOL;
END_VAR

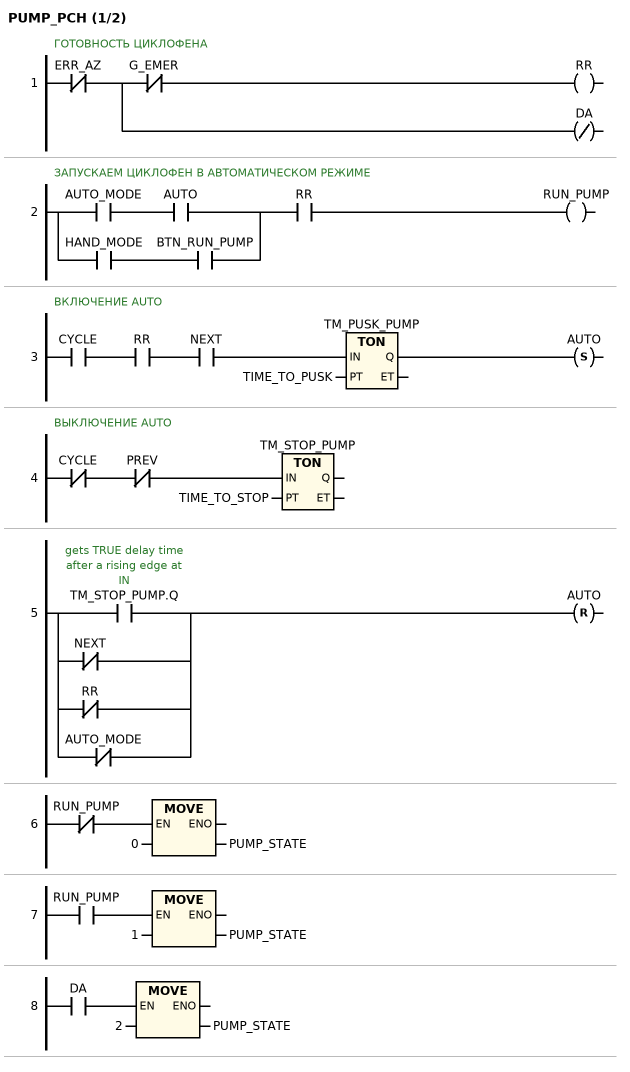
// NETWORK 1
// ГОТОВНОСТЬ ЦИКЛОФЕНА
_w1 := NOT ERR_AZ;
RR := _w1 AND NOT G_EMER;
DA := NOT _w1;

// NETWORK 2
// ЗАПУСКАЕМ ЦИКЛОФЕН В АВТОМАТИЧЕСКОМ РЕЖИМЕ
RUN_PUMP := (AUTO_MODE AND AUTO OR HAND_MODE AND BTN_RUN_PUMP) AND RR;

// NETWORK 3
// ВКЛЮЧЕНИЕ AUTO
TM_PUSK_PUMP(IN := CYCLE AND RR AND NEXT, PT := TIME_TO_PUSK); // TON
AUTO S= TM_PUSK_PUMP.Q;

// NETWORK 4
// ВЫКЛЮЧЕНИЕ AUTO
TM_STOP_PUMP(IN := NOT CYCLE AND NOT PREV, PT := TIME_TO_STOP); // TON

// NETWORK 5
//   TM_STOP_PUMP.Q: gets TRUE delay time after a rising edge at IN
AUTO R= TM_STOP_PUMP.Q OR NOT NEXT OR NOT RR OR NOT AUTO_MODE;

// NETWORK 6
IF NOT RUN_PUMP THEN PUMP_STATE := 0; END_IF

// NETWORK 7
IF RUN_PUMP THEN PUMP_STATE := 1; END_IF

// NETWORK 8
IF DA THEN PUMP_STATE := 2; END_IF

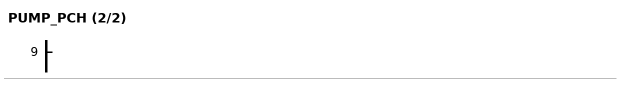
// NETWORK 9

END_FUNCTION_BLOCK

// MyController/Application/POUWER_BOILER
PROGRAM POUWER_BOILER
VAR
	BLINK_RESET_FLOW : BLINK;
	RISE_IMPUT_FLOW : R_TRIG;
	good: BOOL;
	K: REAL;
	TF: REAL;
	POWER_BURNER: REAL;
	//power_utilizator: REAL;
END_VAR

POWER_GRAFIC:=FLOW_GRAFIC*(TMP_PODACHA-TMP_OBRATKA)*99.82/1000000;//Определяем мощность расчетную для котлов

BLINK_RESET_FLOW(ENABLE:=1,TIMELOW:=T#9S,TIMEHIGH:=T#1S);
RISE_IMPUT_FLOW(CLK:=BLINK_RESET_FLOW.OUT);
IF reset_flowmetr.zero_flow=0 AND RISE_IMPUT_FLOW.Q=1 THEN
	power_utilizator:=power_utilizator+FLOW_BOILER_2*(TT7_WTR_IN_2-TT6_WTR_UTIL_IN)*99.82/1000000/360;
END_IF

//fl_g_s:=Qb_s;
//fl_g_l:=Qb_l;
flow_gaz:=Qb_l;
flow_gaz:=SHL(flow_gaz,16);
flow_gaz:=flow_gaz+Qb_s;
V_gaz:=Vb_l;
V_gaz:=SHL(V_gaz,16);
V_gaz:=V_gaz+Vb_s;
//flow_gaz:=flow_gaz*65636;


//	POWER_BOILER_1:=FLOW_BOILER_1*(TT3_WTR_OUT_1-TT2_WTR_IN_1)*99.82/1000000;
//	POWER_BOILER_2:=FLOW_BOILER_2*(TT8_WTR_OUT_2-TT7_WTR_IN_2)*99.82/1000000;

//T_ZADANNOE:= ((POWER_GRAFIC + TT2_WTR_IN_1*(FLOW_BOILER_1+FLOW_BOILER_2))/FLOW_BOILER_1+FLOW_BOILER_2)*(K+(T1_GRAFIC-TF));

//TEMP_POROG_2:= REAL_TO_INT(T_ZADANNOE);

//IF PRIOR_BOILER_1 
//	THEN POWER_BURNER:=1000;
//	ELSE POWER_BURNER:=800;
//END_IF

//POWER_GRAFIC:=FLOW_GRAFIC*(TMP_PODACHA-TMP_OBRATKA);//Определяем мощность расчетную для котлов

//IF POWER_GRAFIC > POWER_BURNER

IF MEDIUM_TEMP_AIR<tmp_use_1_and_2_boiler/10 OR POWER_GRAFIC>=0.95*POWER_BOILER2/1000
	THEN USE_2_BOILERS:=1;
	ELSE USE_2_BOILERS:=0;
END_IF

END_PROGRAM

// MyController/Application/ALL_ERR
PROGRAM ALL_ERR
VAR
	DA_ALL_1: BOOL;
	DA_ALL_2: BOOL;
	DA_ALL_3: BOOL;
	DA_ALL_4: BOOL;
	DA_ALL_5: BOOL;
	DA_ALL_6: BOOL;
	DA_ALL_7: BOOL;
	DA_ALL_8: BOOL;
	DA_ALL_9: BOOL;
	DA_ALL_10: BOOL;
END_VAR

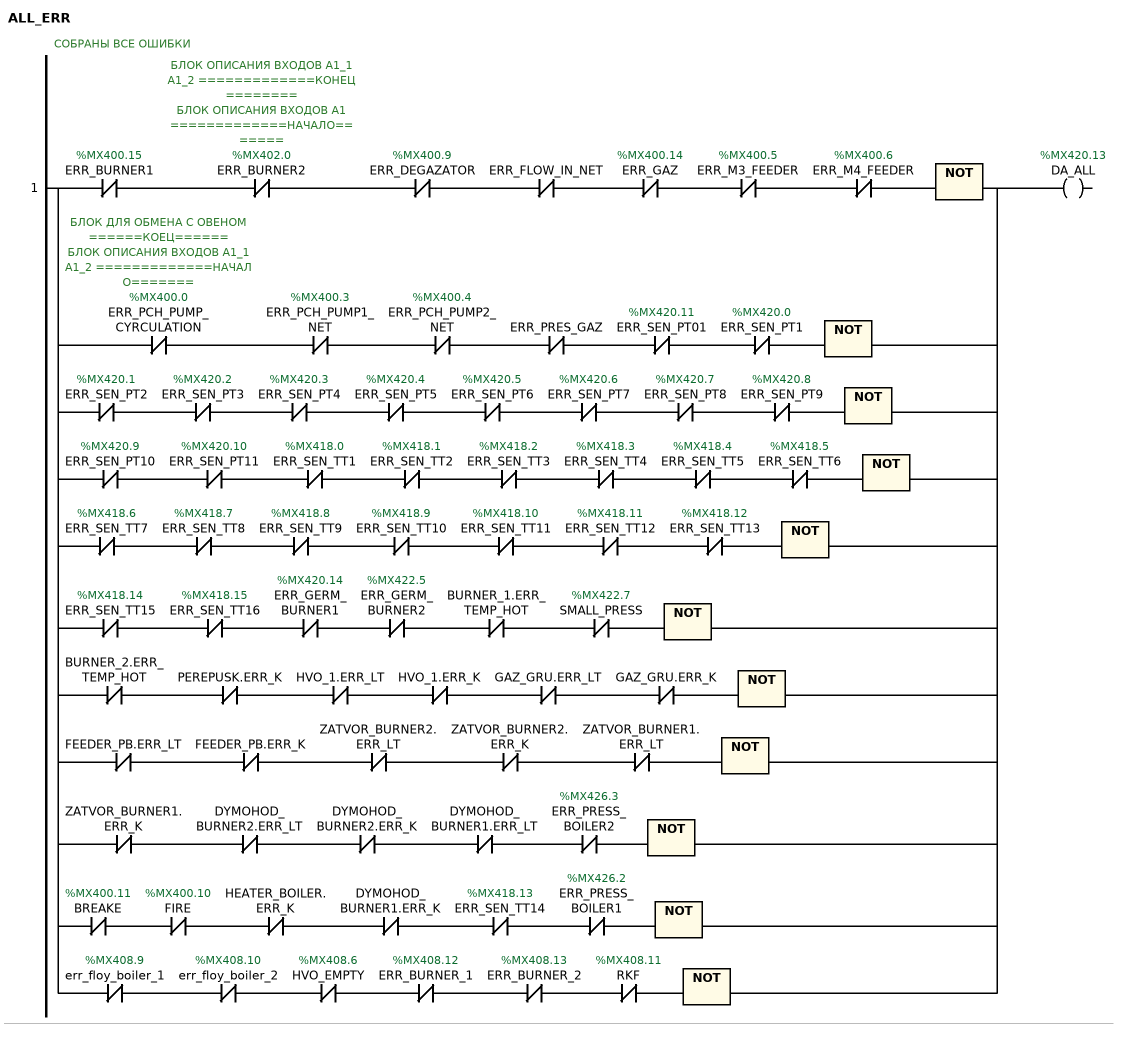
// NETWORK 1
// СОБРАНЫ ВСЕ ОШИБКИ
//   ERR_BURNER1: AT %MX400.15
//   ERR_BURNER2: БЛОК ОПИСАНИЯ ВХОДОВ А1_1 A1_2 =============КОНЕЦ======== БЛОК ОПИСАНИЯ ВХОДОВ А1 =============НАЧАЛО======= | AT %MX402.0
//   ERR_DEGAZATOR: AT %MX400.9
//   ERR_GAZ: AT %MX400.14
//   ERR_M3_FEEDER: AT %MX400.5
//   ERR_M4_FEEDER: AT %MX400.6
//   ERR_PCH_PUMP_CYRCULATION: БЛОК ДЛЯ ОБМЕНА С ОВЕНОМ ======КОЕЦ====== БЛОК ОПИСАНИЯ ВХОДОВ А1_1 A1_2 =============НАЧАЛО======= | AT %MX400.0
//   ERR_PCH_PUMP1_NET: AT %MX400.3
//   ERR_PCH_PUMP2_NET: AT %MX400.4
//   ERR_SEN_PT01: AT %MX420.11
//   ERR_SEN_PT1: AT %MX420.0
//   ERR_SEN_PT2: AT %MX420.1
//   ERR_SEN_PT3: AT %MX420.2
//   ERR_SEN_PT4: AT %MX420.3
//   ERR_SEN_PT5: AT %MX420.4
//   ERR_SEN_PT6: AT %MX420.5
//   ERR_SEN_PT7: AT %MX420.6
//   ERR_SEN_PT8: AT %MX420.7
//   ERR_SEN_PT9: AT %MX420.8
//   ERR_SEN_PT10: AT %MX420.9
//   ERR_SEN_PT11: AT %MX420.10
//   ERR_SEN_TT1: AT %MX418.0
//   ERR_SEN_TT2: AT %MX418.1
//   ERR_SEN_TT3: AT %MX418.2
//   ERR_SEN_TT4: AT %MX418.3
//   ERR_SEN_TT5: AT %MX418.4
//   ERR_SEN_TT6: AT %MX418.5
//   ERR_SEN_TT7: AT %MX418.6
//   ERR_SEN_TT8: AT %MX418.7
//   ERR_SEN_TT9: AT %MX418.8
//   ERR_SEN_TT10: AT %MX418.9
//   ERR_SEN_TT11: AT %MX418.10
//   ERR_SEN_TT12: AT %MX418.11
//   ERR_SEN_TT13: AT %MX418.12
//   ERR_SEN_TT15: AT %MX418.14
//   ERR_SEN_TT16: AT %MX418.15
//   ERR_GERM_BURNER1: AT %MX420.14
//   ERR_GERM_BURNER2: AT %MX422.5
//   SMALL_PRESS: AT %MX422.7
//   ERR_PRESS_BOILER2: AT %MX426.3
//   BREAKE: AT %MX400.11
//   FIRE: AT %MX400.10
//   ERR_SEN_TT14: AT %MX418.13
//   ERR_PRESS_BOILER1: AT %MX426.2
//   err_floy_boiler_1: AT %MX408.9
//   err_floy_boiler_2: AT %MX408.10
//   HVO_EMPTY: AT %MX408.6
//   ERR_BURNER_1: AT %MX408.12
//   ERR_BURNER_2: AT %MX408.13
//   RKF: AT %MX408.11
//   DA_ALL: AT %MX420.13
DA_ALL := NOT (NOT ERR_BURNER1 AND NOT ERR_BURNER2 AND NOT ERR_DEGAZATOR AND NOT ERR_FLOW_IN_NET AND NOT ERR_GAZ AND NOT ERR_M3_FEEDER AND NOT ERR_M4_FEEDER) OR NOT (NOT ERR_PCH_PUMP_CYRCULATION AND NOT ERR_PCH_PUMP1_NET AND NOT ERR_PCH_PUMP2_NET AND NOT ERR_PRES_GAZ AND NOT ERR_SEN_PT01 AND NOT ERR_SEN_PT1) OR NOT (NOT ERR_SEN_PT2 AND NOT ERR_SEN_PT3 AND NOT ERR_SEN_PT4 AND NOT ERR_SEN_PT5 AND NOT ERR_SEN_PT6 AND NOT ERR_SEN_PT7 AND NOT ERR_SEN_PT8 AND NOT ERR_SEN_PT9) OR NOT (NOT ERR_SEN_PT10 AND NOT ERR_SEN_PT11 AND NOT ERR_SEN_TT1 AND NOT ERR_SEN_TT2 AND NOT ERR_SEN_TT3 AND NOT ERR_SEN_TT4 AND NOT ERR_SEN_TT5 AND NOT ERR_SEN_TT6) OR NOT (NOT ERR_SEN_TT7 AND NOT ERR_SEN_TT8 AND NOT ERR_SEN_TT9 AND NOT ERR_SEN_TT10 AND NOT ERR_SEN_TT11 AND NOT ERR_SEN_TT12 AND NOT ERR_SEN_TT13) OR NOT (NOT ERR_SEN_TT15 AND NOT ERR_SEN_TT16 AND NOT ERR_GERM_BURNER1 AND NOT ERR_GERM_BURNER2 AND NOT BURNER_1.ERR_TEMP_HOT AND NOT SMALL_PRESS) OR NOT (NOT BURNER_2.ERR_TEMP_HOT AND NOT PEREPUSK.ERR_K AND NOT HVO_1.ERR_LT AND NOT HVO_1.ERR_K AND NOT GAZ_GRU.ERR_LT AND NOT GAZ_GRU.ERR_K) OR NOT (NOT FEEDER_PB.ERR_LT AND NOT FEEDER_PB.ERR_K AND NOT ZATVOR_BURNER2.ERR_LT AND NOT ZATVOR_BURNER2.ERR_K AND NOT ZATVOR_BURNER1.ERR_LT) OR NOT (NOT ZATVOR_BURNER1.ERR_K AND NOT DYMOHOD_BURNER2.ERR_LT AND NOT DYMOHOD_BURNER2.ERR_K AND NOT DYMOHOD_BURNER1.ERR_LT AND NOT ERR_PRESS_BOILER2) OR NOT (NOT BREAKE AND NOT FIRE AND NOT HEATER_BOILER.ERR_K AND NOT DYMOHOD_BURNER1.ERR_K AND NOT ERR_SEN_TT14 AND NOT ERR_PRESS_BOILER1) OR NOT (NOT err_floy_boiler_1 AND NOT err_floy_boiler_2 AND NOT HVO_EMPTY AND NOT ERR_BURNER_1 AND NOT ERR_BURNER_2 AND NOT RKF);

END_PROGRAM

// MyController/Application/zadanie_for_burner
PROGRAM zadanie_for_burner
VAR
	FLOW_SUM: INT;
	BLINKER : BLINK;
	RTRIGInst : R_TRIG; 
	day: BOOL;
	k1: REAL;
END_VAR

VAR_INPUT
	
END_VAR

//Каждые TIMELOW минут смотри темературу на улице и корректируем задание для горелок
BLINKER(ENABLE:=1,TIMELOW:=T#30M,TIMEHIGH:=T#2S);
RTRIGInst(CLK:=BLINKER.OUT); 
IF RTRIGInst.Q=1 THEN
	MEDIUM_TEMP_AIR:=(TT16_ON_AIR/10);
END_IF

//Смотрим на температуру наружнего воздуха и берем из массива температуру для горелок 
IF (MEDIUM_TEMP_AIR)>-25 AND (MEDIUM_TEMP_AIR)<11
THEN 
	TMP_PODACHA:=T_graf_1[10-MEDIUM_TEMP_AIR];
	TMP_OBRATKA:=T_graf_2[10-MEDIUM_TEMP_AIR];	
ELSE
	IF MEDIUM_TEMP_AIR >= 11 THEN
		TMP_PODACHA:=T_graf_1[0];
		TMP_OBRATKA:=T_graf_2[0];
	END_IF
	IF MEDIUM_TEMP_AIR <=-25 THEN
		TMP_PODACHA:=T_graf_1[34];
		TMP_OBRATKA:=T_graf_2[34];
	END_IF
END_IF

IF day=FALSE AND day_mode.uiGetHour>=DayModeHourStart AND day_mode.uiGetMinute>=DayModeMinuteStart  
 THEN
	day:=TRUE;	
END_IF

IF day=TRUE AND day_mode.uiGetHour>=DayModeHourStop AND day_mode.uiGetMinute>=DayModeMinuteStop
 THEN
	day:=FALSE;		
END_IF

IF day AND MEDIUM_TEMP_AIR >= DayModeTempAir/10 THEN
	TMP_PODACHA:=DayModeTempWater;
END_IF
k1:=INT_TO_REAL(K);
k1:=k1/100;
FLOW_SUM:=REAL_TO_INT(FLOW_BOILER_1+FLOW_BOILER_2);//Расход через два котла
IF use_balanse_power=TRUE AND FLOW_SUM>0
	THEN
		POWER_GRAFIC:=FLOW_GRAFIC*(TMP_PODACHA-TMP_OBRATKA);//Определяем мощность расчетную для котлов
		ZADANIE_BALANSE:=REAL_TO_INT((((POWER_GRAFIC+TT13_NET_WTR_IN2*FLOW_SUM)*(k1))/(FLOW_SUM+1)) + (TMP_PODACHA-TT12_NET_WTR_OUT));

		IF ZADANIE_BALANSE > MAX_TEMP_BALANSE THEN ZADANIE_BALANSE:= MAX_TEMP_BALANSE;
		END_IF
	ELSE
		ZADANIE_TMP_BURNER_1:=MANUAL_ZADANIE_TMP_BURNER1;
		ZADANIE_TMP_BURNER_2:=MANUAL_ZADANIE_TMP_BURNER2;
END_IF

//ZADANIE_TMP_BURNER_2:=ZADANIE_TMP_BURNER_1;

//Задание для трехходового клапана перепуска
IF PEREPUSK_AUTO=1
	THEN 
		TT12_NET_WATER_ZADANIE:=TMP_PODACHA;
	ELSE 
		TT12_NET_WATER_ZADANIE:=ManZadaniePerepusk;
END_IF



IF BURNER1_AUTO=1 AND use_balanse_power=TRUE
	THEN ZADANIE_TMP_BURNER_1:=ZADANIE_BALANSE_AVG;
	ELSE ZADANIE_TMP_BURNER_1:=MANUAL_ZADANIE_TMP_BURNER1;
END_IF

IF BURNER2_AUTO=1 AND use_balanse_power=TRUE
	THEN ZADANIE_TMP_BURNER_2:=ZADANIE_BALANSE_AVG;
	ELSE ZADANIE_TMP_BURNER_2:=MANUAL_ZADANIE_TMP_BURNER2;
END_IF

END_PROGRAM

// MyController/Application/set_time
PROGRAM set_time
VAR
      udiResultConvertToUtc: UDINT; 
      dwSetTimeStamp: DWORD;

      uidResultRtcSet: UDINT;
	  set_time: TON;
END_VAR
VAR // added by the converter: edge detectors and wires of the graphical bodies
    _s1 : RTS_SYSTIMEDATE;
    _w1, _w4 : BOOL;
    _w2, _w3 : ANY;
END_VAR

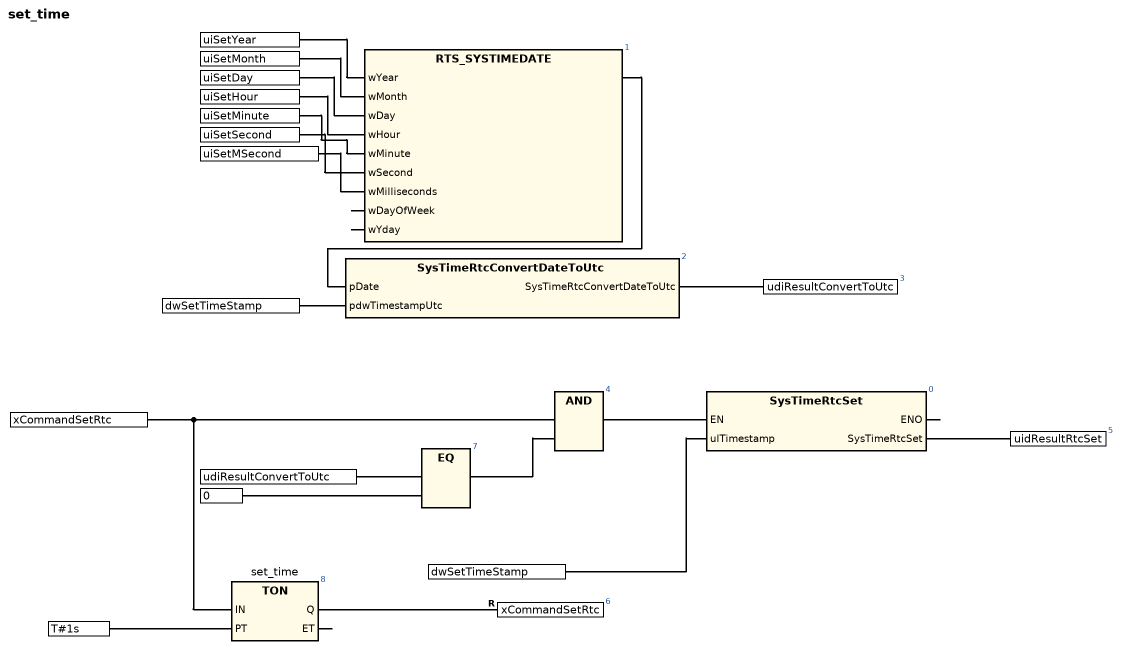
IF _w1 THEN _w2 := SysTimeRtcSet(ulTimestamp := dwSetTimeStamp); END_IF
// compose _s1 : RTS_SYSTIMEDATE
_s1.wYear := uiSetYear;
_s1.wMonth := uiSetMonth;
_s1.wDay := uiSetDay;
_s1.wHour := uiSetHour;
_s1.wMinute := uiSetMinute;
_s1.wSecond := uiSetSecond;
_s1.wMilliseconds := uiSetMSecond;
_w3 := SysTimeRtcConvertDateToUtc(pDate := _s1, pdwTimestampUtc := dwSetTimeStamp);
udiResultConvertToUtc := _w3;
_w1 := xCommandSetRtc AND _w4;
uidResultRtcSet := _w2;
xCommandSetRtc R= set_time.Q;
_w4 := udiResultConvertToUtc = 0;
set_time(IN := xCommandSetRtc, PT := T#1s); // TON

END_PROGRAM

// MyController/Application/ERR_SENSER
PROGRAM ERR_SENSER
VAR
	ERR_PT: INT;
END_VAR

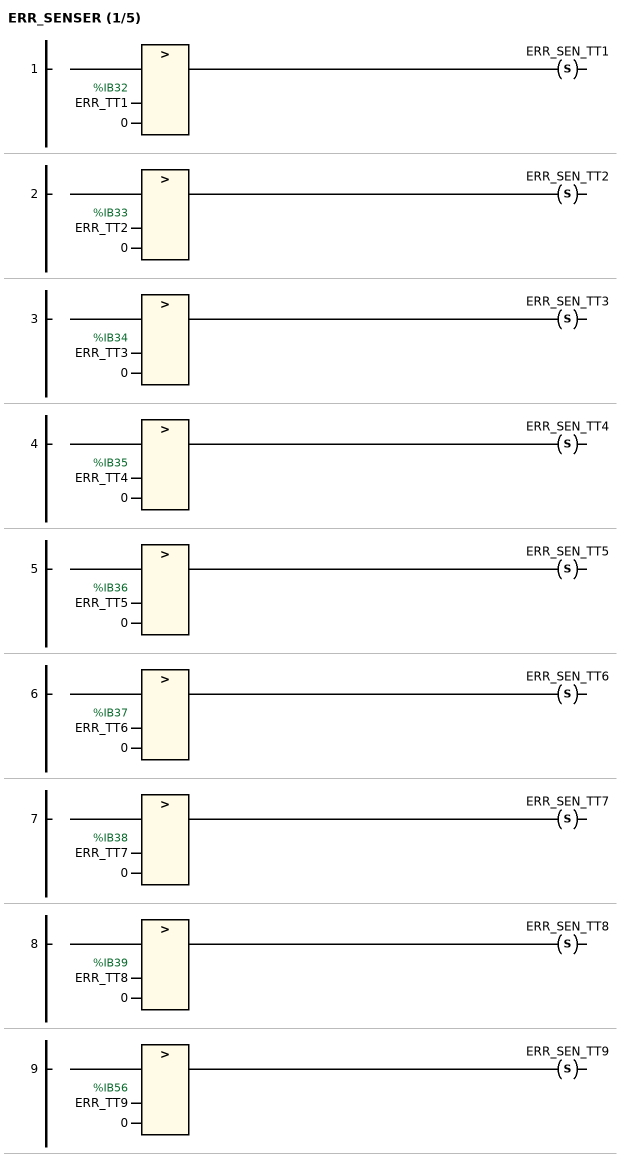
// NETWORK 1
//   ERR_TT1: A1_4 : | AT %IB32
ERR_SEN_TT1 S= ERR_TT1 > 0;

// NETWORK 2
//   ERR_TT2: A1_4 : | AT %IB33
ERR_SEN_TT2 S= ERR_TT2 > 0;

// NETWORK 3
//   ERR_TT3: A1_4 : | AT %IB34
ERR_SEN_TT3 S= ERR_TT3 > 0;

// NETWORK 4
//   ERR_TT4: A1_4 : | AT %IB35
ERR_SEN_TT4 S= ERR_TT4 > 0;

// NETWORK 5
//   ERR_TT5: A1_4 : | AT %IB36
ERR_SEN_TT5 S= ERR_TT5 > 0;

// NETWORK 6
//   ERR_TT6: A1_4 : | AT %IB37
ERR_SEN_TT6 S= ERR_TT6 > 0;

// NETWORK 7
//   ERR_TT7: A1_4 : | AT %IB38
ERR_SEN_TT7 S= ERR_TT7 > 0;

// NETWORK 8
//   ERR_TT8: A1_4 : | AT %IB39
ERR_SEN_TT8 S= ERR_TT8 > 0;

// NETWORK 9
//   ERR_TT9: A1_5 : | AT %IB56
ERR_SEN_TT9 S= ERR_TT9 > 0;

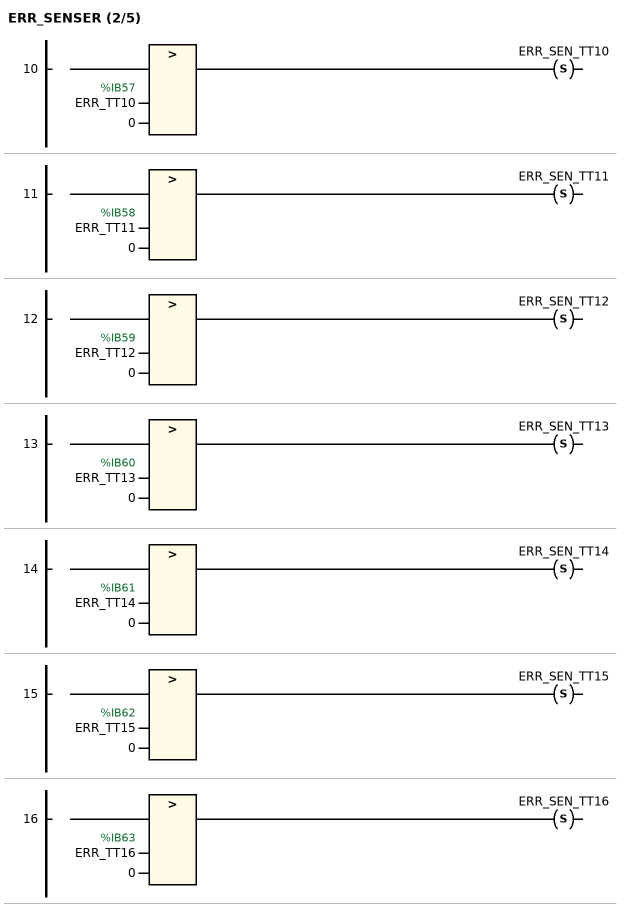
// NETWORK 10
//   ERR_TT10: A1_5 : | AT %IB57
ERR_SEN_TT10 S= ERR_TT10 > 0;

// NETWORK 11
//   ERR_TT11: A1_5 : | AT %IB58
ERR_SEN_TT11 S= ERR_TT11 > 0;

// NETWORK 12
//   ERR_TT12: A1_5 : | AT %IB59
ERR_SEN_TT12 S= ERR_TT12 > 0;

// NETWORK 13
//   ERR_TT13: A1_5 : | AT %IB60
ERR_SEN_TT13 S= ERR_TT13 > 0;

// NETWORK 14
//   ERR_TT14: A1_5 : | AT %IB61
ERR_SEN_TT14 S= ERR_TT14 > 0;

// NETWORK 15
//   ERR_TT15: A1_5 : | AT %IB62
ERR_SEN_TT15 S= ERR_TT15 > 0;

// NETWORK 16
//   ERR_TT16: A1_5 : | AT %IB63
ERR_SEN_TT16 S= ERR_TT16 > 0;

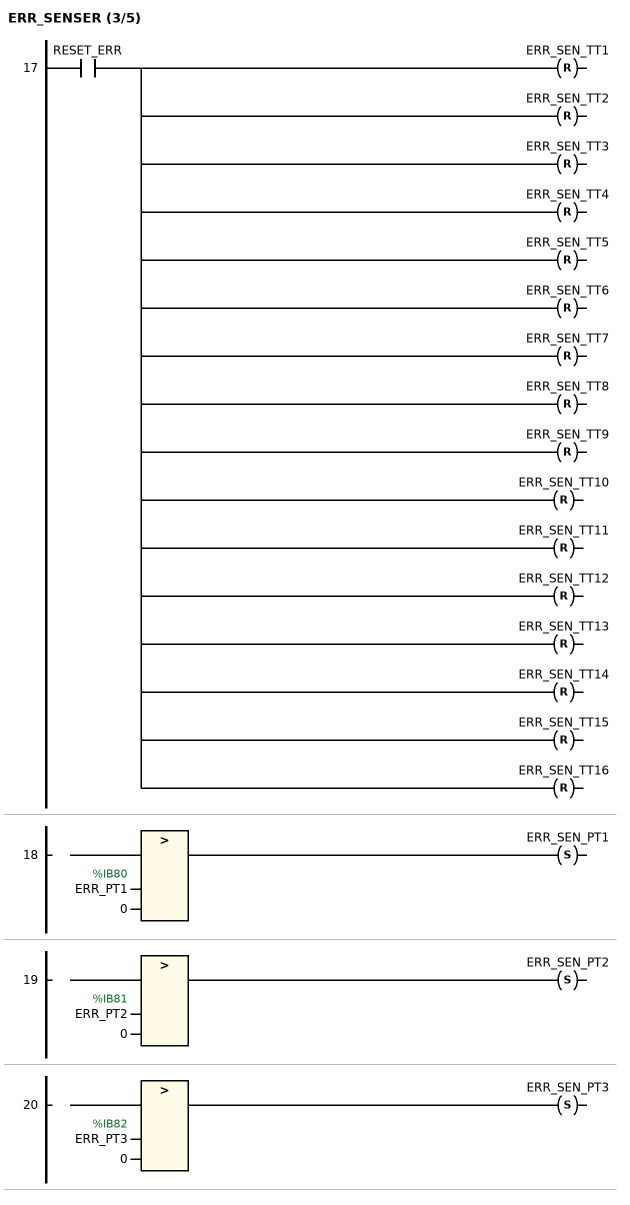
// NETWORK 17
ERR_SEN_TT1 R= RESET_ERR;
ERR_SEN_TT2 R= RESET_ERR;
ERR_SEN_TT3 R= RESET_ERR;
ERR_SEN_TT4 R= RESET_ERR;
ERR_SEN_TT5 R= RESET_ERR;
ERR_SEN_TT6 R= RESET_ERR;
ERR_SEN_TT7 R= RESET_ERR;
ERR_SEN_TT8 R= RESET_ERR;
ERR_SEN_TT9 R= RESET_ERR;
ERR_SEN_TT10 R= RESET_ERR;
ERR_SEN_TT11 R= RESET_ERR;
ERR_SEN_TT12 R= RESET_ERR;
ERR_SEN_TT13 R= RESET_ERR;
ERR_SEN_TT14 R= RESET_ERR;
ERR_SEN_TT15 R= RESET_ERR;
ERR_SEN_TT16 R= RESET_ERR;

// NETWORK 18
//   ERR_PT1: A1_6 : | AT %IB80
ERR_SEN_PT1 S= ERR_PT1 > 0;

// NETWORK 19
//   ERR_PT2: A1_6 : | AT %IB81
ERR_SEN_PT2 S= ERR_PT2 > 0;

// NETWORK 20
//   ERR_PT3: A1_6 : | AT %IB82
ERR_SEN_PT3 S= ERR_PT3 > 0;

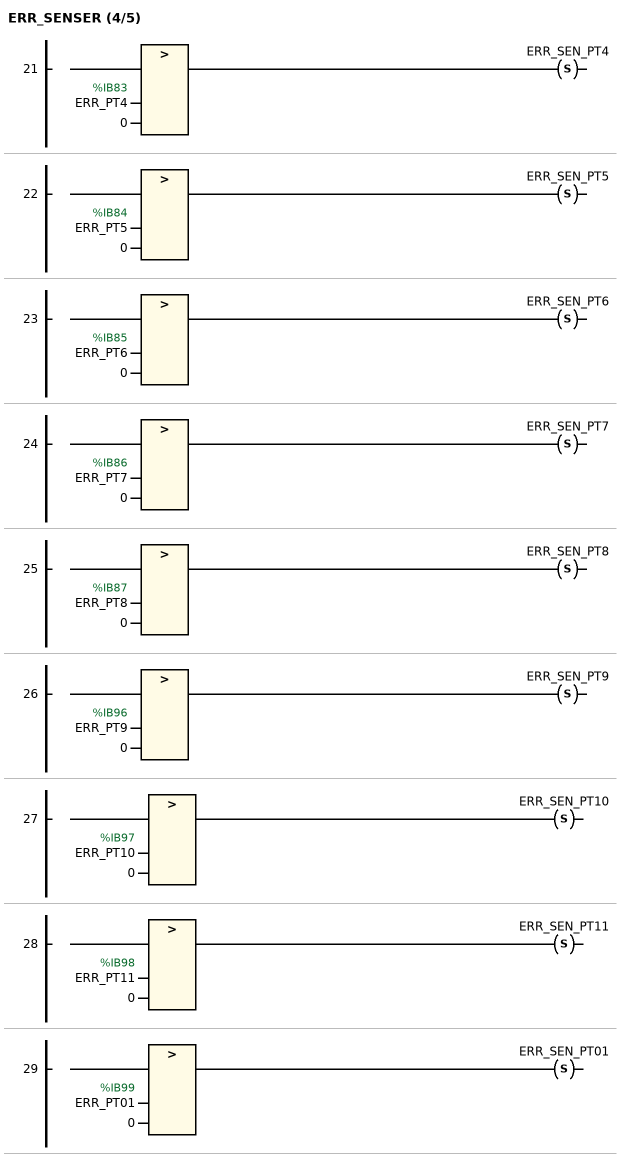
// NETWORK 21
//   ERR_PT4: A1_6 : | AT %IB83
ERR_SEN_PT4 S= ERR_PT4 > 0;

// NETWORK 22
//   ERR_PT5: A1_6 : | AT %IB84
ERR_SEN_PT5 S= ERR_PT5 > 0;

// NETWORK 23
//   ERR_PT6: A1_6 : | AT %IB85
ERR_SEN_PT6 S= ERR_PT6 > 0;

// NETWORK 24
//   ERR_PT7: A1_6 : | AT %IB86
ERR_SEN_PT7 S= ERR_PT7 > 0;

// NETWORK 25
//   ERR_PT8: A1_6 : | AT %IB87
ERR_SEN_PT8 S= ERR_PT8 > 0;

// NETWORK 26
//   ERR_PT9: A1_7 : | AT %IB96
ERR_SEN_PT9 S= ERR_PT9 > 0;

// NETWORK 27
//   ERR_PT10: A1_7 : | AT %IB97
ERR_SEN_PT10 S= ERR_PT10 > 0;

// NETWORK 28
//   ERR_PT11: A1_7 : | AT %IB98
ERR_SEN_PT11 S= ERR_PT11 > 0;

// NETWORK 29
//   ERR_PT01: A1_7 : | AT %IB99
ERR_SEN_PT01 S= ERR_PT01 > 0;

